// Mitsubishi GX Works2 project: Operacoes_function_03.10   PLC: Q03UDV

// task Task_01 (event TRUE, interval 0, priority 31): POU_01
// task ST_Example (event TRUE, interval 0, priority 31): ST_Example

PROGRAM POU_01
VAR
  IntMult : ARRAY [0..1] OF DINT;
  fbBlinker_Test : fbBlinker;
  fbBlinkerTes : fbBlinker;
  fbBlinkerTest : fbBlinker;
  result : DINT;
  Divresult : ARRAY [0..1] OF INT;
END_VAR
(* structured ladder/FBD written out as ST: instructions are called as NAME(EN, inputs, outputs); _pN, _eN, _tN stand for wires *)
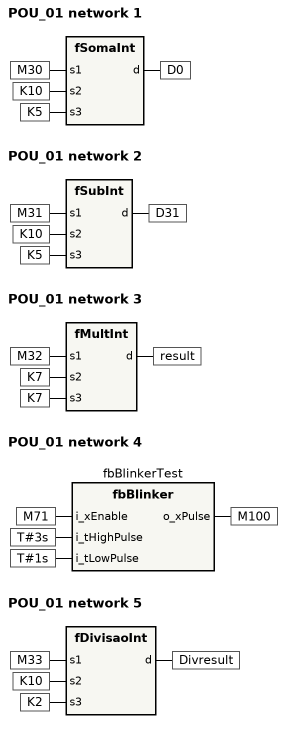
(* network 1 *)
D0 := fSomaInt(M30, K10, K5);
(* network 2 *)
D31 := fSubInt(M31, K10, K5);
(* network 3 *)
result := fMultInt(M32, K7, K7);
(* network 4 *)
fbBlinkerTest(i_xEnable := M71, i_tHighPulse := T#3s, i_tLowPulse := T#1s, o_xPulse => M100);
(* network 5 *)
Divresult := fDivisaoInt(M33, K10, K2);
END_PROGRAM

FUNCTION fSomaInt
VAR_INPUT
  i_xHabilitar : BOOL;
  i_iElemento1 : INT;
  i_iElemento2 : INT;
END_VAR
(* structured ladder/FBD written out as ST: instructions are called as NAME(EN, inputs, outputs); _pN, _eN, _tN stand for wires *)
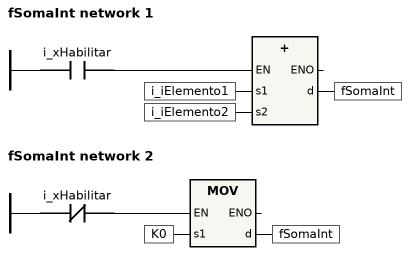
(* network 1 *)
+(i_xHabilitar, i_iElemento1, i_iElemento2, fSomaInt);
(* network 2 *)
MOV(NOT i_xHabilitar, K0, fSomaInt);
END_FUNCTION

FUNCTION fSubInt
VAR_INPUT
  i_xSub : BOOL;
  i_iNum1 : INT;
  i_iNum2 : INT;
END_VAR
(* structured ladder/FBD written out as ST: instructions are called as NAME(EN, inputs, outputs); _pN, _eN, _tN stand for wires *)
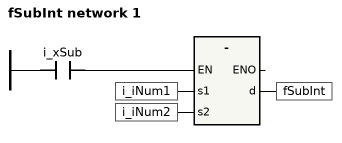
(* network 1 *)
-(i_xSub, i_iNum1, i_iNum2, fSubInt);
END_FUNCTION

FUNCTION_BLOCK fbBlinker
VAR_INPUT
  i_xEnable : BOOL;
  i_tHighPulse : TIME;
  i_tLowPulse : TIME;
END_VAR
VAR_OUTPUT
  o_xPulse : BOOL;
END_VAR
VAR
  fbTimerHigh : TP;
  fbTimerLow : TOF;
  xAuxiliar : BOOL;
  TP_1 : TP;
  TOF_1 : TOF;
END_VAR
(* structured ladder/FBD written out as ST: instructions are called as NAME(EN, inputs, outputs); _pN, _eN, _tN stand for wires *)
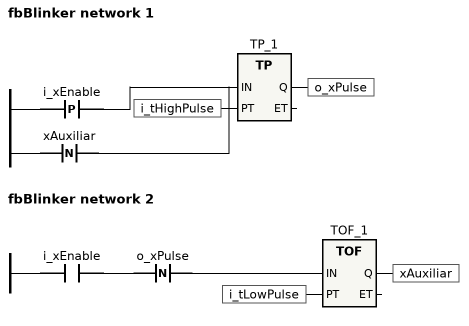
(* network 1 *)
TP_1(IN := LDP(TRUE, i_xEnable) OR LDF(TRUE, xAuxiliar), PT := i_tHighPulse, Q => o_xPulse);
(* network 2 *)
TOF_1(IN := i_xEnable AND LDF(TRUE, o_xPulse), PT := i_tLowPulse, Q => xAuxiliar);
END_FUNCTION_BLOCK

FUNCTION fMultInt
VAR_INPUT
  i_xMultInt : BOOL;
  i_iNum4 : INT;
  i_iNum3 : INT;
END_VAR
(* structured ladder/FBD written out as ST: instructions are called as NAME(EN, inputs, outputs); _pN, _eN, _tN stand for wires *)
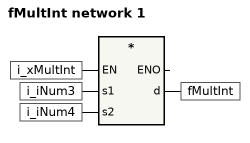
(* network 1 *)
*(i_xMultInt, i_iNum3, i_iNum4, fMultInt);
END_FUNCTION

FUNCTION fDivisaoInt
VAR_INPUT
  i_xFuncDiv : BOOL;
  i_iNum5 : INT;
  i_iNum6 : INT;
END_VAR
(* structured ladder/FBD written out as ST: instructions are called as NAME(EN, inputs, outputs); _pN, _eN, _tN stand for wires *)
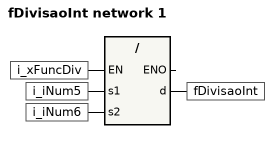
(* network 1 *)
/(i_xFuncDiv, i_iNum5, i_iNum6, fDivisaoInt);
END_FUNCTION

PROGRAM ST_Example
VAR
  iDR : ARRAY [0..99] OF INT;  (* Declaração de variável ST *)
END_VAR
VAR CONSTANT
  iEle01 : INT := 15;  (* Elemento 01 de operação *)
  iEle02 : INT := 4;  (* Elemento 02 de operação *)
END_VAR
VAR
  iArrayTest : INT;
  fBlinkerTestST : fbBlinker;  (* Declaração de variável ST *)
  fBTPTestST : TP;  (* Declaração de variável ST *)
  fSomaInt : ARRAY [0..4] OF INT;
  iValidarvalor : INT;
  iContador : INT;
END_VAR


iDR[0] := iEle01 + iEle02;
iDR[1] := iEle01 - iEle02;
iDR[2] := iEle01 * iEle02;
iDR[3] := iEle01 / iEle02;



fBlinkerTestST(i_xEnable:= M35 ,i_tHighPulse:= T#2s ,i_tLowPulse:= T#500ms ,o_xPulse:= Y35 );
(*fBTPTestST(IN:= ?BOOL? ,PT:= ?TIME? ,Q:= ?BOOL? ,ET:= ?TIME? );*)


iDR[4] :=  fSomaST( 100 , 2 );
iDR[5] := fSub (100, 50);
iDR[6] := fMultST( 15 , 3 );
iDR[7] := fDivST( 100 , 10 );



(*IF  ?condition?  THEN
	 ?statement? ;
ELSE
	 ?statement? ;
END_IF;  *)


(*CASE  iValidarvalor OF
	 0,10 :
		iDR[0] := iEle01 + iEle02 ;
	 1,11 :
		 iDR[0] := iEle01 - iEle02;
	 ?value 3? :
		 ?statement? ;
	ELSE
		 ?statement? ;
END_CASE;*)
	
IF iContador <= 12 THEN	
	FOR iContador := 0  TO  6  BY  1  DO
	 	iDR[iContador] := iContador+2;
	END_FOR;
END_IF;
END_PROGRAM

FUNCTION fSomaST
VAR_INPUT
  i_Num1 : INT;
  i_Num2 : INT;
END_VAR
fSomaST := i_Num1+i_Num2;
END_FUNCTION

FUNCTION fSub
VAR_INPUT
  i_Num3 : INT;
  i_Num4 : INT;
END_VAR

fSub := i_Num3 - i_Num4;
END_FUNCTION

FUNCTION fMultST
VAR_INPUT
  i_Num5 : INT;
  i_Num6 : INT;
END_VAR
fMultST := i_Num5 * i_Num6;
END_FUNCTION

FUNCTION fDivST
VAR_INPUT
  i_Num7 : INT;
  i_Num8 : INT;
END_VAR
fDivST := i_Num7 / i_Num8;
END_FUNCTION

FUNCTION_BLOCK fbOperacoesST
VAR_INPUT
  i_Operacoes : ARRAY [0..99] OF INT;
END_VAR

;
END_FUNCTION_BLOCK
